(* Logix 5000 project; controller OptixTest vendor 1 type 14 code 194 rev 38.11; software revision 38.01 *)

TASK MainTask (continuous, watchdog 500 ms) : MainProgram

MODULES
   Local : vendor 1 type 14 code 194 (5069 0, rev 38.11)
END_MODULES

TYPE MyUDT :
STRUCT
   MySTRING : STRING;
   MyDINT : DINT;
   MyREAL : REAL;
   MyBOOL : BOOL;
END_STRUCT
END_TYPE

VAR_GLOBAL   (* controller tags *)
   MyUDTArray : MyUDT[10] := ([0].MySTRING := 'Index 0', [1].MySTRING := 'Index 1', [1].MyDINT := 1, [1].MyREAL := 1.0, [1].MyBOOL := 1, [2].MySTRING := 'Index 2', [2].MyDINT := 2, [2].MyREAL := 2.0, [3].MySTRING := 'Index 3', [3].MyDINT := 3, [3].MyREAL := 3.0, [3].MyBOOL := 1, [4].MySTRING := 'Index 4', [4].MyDINT := 4, [4].MyREAL := 4.0, [5].MySTRING := 'Index 5', [5].MyDINT := 5, [5].MyREAL := 5.0, [5].MyBOOL := 1, [6].MySTRING := 'Index 6', [6].MyDINT := 6, [6].MyREAL := 6.0, [7].MySTRING := 'Index 7', [7].MyDINT := 7, [7].MyREAL := 7.0, [7].MyBOOL := 1, [8].MySTRING := 'Index 8', [8].MyDINT := 8, [8].MyREAL := 8.0, [9].MySTRING := 'Index 9', [9].MyDINT := 9, [9].MyREAL := 9.0, [9].MyBOOL := 1);
END_VAR

PROGRAM MainProgram   (* main routine MainRoutine *)

ROUTINE MainRoutine   (* ladder *)
END_ROUTINE
END_PROGRAM
